FUNCTION_BLOCK Q_Size (* Command change size ( Part 6 - F.18 ) *)
  (* Standard: ISO 11783-6; Description: Copyright (c) 2022 HR Agrartechnik GmbH This program and the accompanying materials are made available under the terms of the Eclipse Public License 2.0 which is available at https://www.eclipse.org/legal/epl-2.0/ SPDX-License-Identifier: EPL-2.0 see Description Tab *)
  (* Version 1.2, 2026-09-05, Franz Höpfinger, HR Agrartechnik GmbH, Implement xScale scaling multiply *)
  (* Version 1.1, 2026-09-05, Franz Höpfinger, HR Agrartechnik GmbH, Add xScale flag *)
  (* Version 1.0, 2022-07-08, Franz Höpfinger, HR Agrartechnik GmbH *)
  PACKAGE isobus::UT::Q;
  IMPORT isobus::UT::Q::const::IDs::ID_NULL;
  (* Documentation:
  Command change size  ( Part 6 - F.18 )
   The Change Size command is used to change the size of an object. A value of 0 for width or height (or both) means that the object size is 0 and the object is not drawn (Annex F.18). The command targets objects that have the sizeable attribute.
   Valid Object IDs
   A sizeable Object ID is valid if it falls within one of the following ISO 11783-6 ID ranges:
    - Container: 3000 – 3999
   - Button: 6000 – 6999
   - InputBooleanField: 7000 – 7999
   - InputStringField: 8000 – 8999
   - InputNumberField: 9000 – 9999
   - InputListField: 10000 – 10999
   - OutputStringField: 11000 – 11999
   - OutputNumberField: 12000 – 12999
   - TypLine: 13000 – 13999
   - TypRectangle: 14000 – 14999
   - TypEllipse: 15000 – 15999
   - TypPolygon: 16000 – 16999
   - Meter: 17000 – 17999
   - LinearBarGraph: 18000 – 18999
   - ArchedBarGraph: 19000 – 19999
   - OutputListObject: 37000 – 37999
   - AnimationObject: 44000 – 44999
    ID_NULL (65535) is not a command target but can be used in INIT to deactivate the FB. Any ID outside these ranges is invalid for commanding.
   Activate / Deactivate
   The FB is deactivated by default. It becomes active when INIT provides a valid sizeable Object ID. Sending INIT with ID_NULL (65535) deactivates the FB again. This toggle can be repeated arbitrarily.
    - INIT + ID_NULL (65535): FB deactivated, STATUS="DEACTIVATED", s16result=VT_E_DEACTIVATED (-40)
   - INIT + valid sizeable ID: FB activated, STATUS="initialized", s16result=VT_E_NO_ERR (0). If a REQ was buffered before, it is executed immediately.
   - INIT + invalid ID: STATUS="ERROR: Invalid Object ID (not a sizeable object)", s16result=VT_E_INVALID_OBJECT_ID (-132)
    REQ Handling
    - REQ before any INIT: Buffered, STATUS="Buffered: INIT not yet completed", s16result=VT_E_NOT_READY (-131)
   - REQ while deactivated (INIT came with NULL or invalid ID): STATUS shows the actual deactivation reason, s16result=VT_E_DEACTIVATED (-40) or VT_E_INVALID_OBJECT_ID (-132)
   - REQ while active: Command sent to VT, result reflected in CNF
    param[in] {objectID, uint16_t}
   Object ID. Use ID_NULL (65535) to deactivate the FB. Use a valid sizeable object ID to activate.
   param[in] {newWidth, uint16_t}
   New width
   param[in] {newHeight, uint16_t}
   New height
   Return Values (s16result):
   int16_t
    - VT_E_NO_ERR (0) - OK
   - VT_E_DEACTIVATED (-40) - FB deactivated (INIT received with ID_NULL)
   - VT_E_INVALID_OBJECT_ID (-132) - Object ID is invalid (not a sizeable object)
   - VT_E_NOT_READY (-131) - Buffered: INIT not yet completed
   - VT_E_OVERFLOW (-6) - buffer overflow
   - VT_E_NOACT (-8) - Command not possible in current state
   - VT_E_NO_INSTANCE (-21) - No VT client available
   - VT_E_ISO_INSTANCE_INVALID (-129) - Identifier for instance (connection) invalid
   - VT_E_NOT_ALIVE (-130) - Identifier for instance valid, but VT Dead.
    Instanz-Eindeutigkeit (Instance Uniqueness)
   Dieser Baustein erfordert Instanz-Eindeutigkeit bezüglich u16ObjId. Es darf im gesamten Programm nur eine Instanz von Q_Size für dieselbe Ziel-Objekt-ID existieren. Eine zweite Instanz auf dieselbe Objekt-ID wird bei INIT deaktiviert (STATUS = "This objID is already in use").
  *)
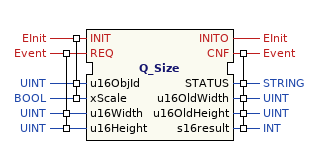
  EVENT_INPUT
    INIT : EInit WITH u16ObjId, xScale; (* Service Initialization *)
    REQ WITH u16Width, u16Height; (* Service Request *)
  END_EVENT
  EVENT_OUTPUT
    INITO : EInit; (* Initialization Confirm *)
    CNF WITH STATUS, s16result, u16OldWidth, u16OldHeight; (* Confirmation of Requested Service *)
  END_EVENT
  VAR_INPUT
    u16ObjId : UINT := ID_NULL; (* Object ID *)
    xScale : BOOL := FALSE; (* FALSE (default) = bypass, send u16Width/u16Height through unchanged. TRUE = scale them by the DM/SKM factor for u16ObjId. *)
    u16Width : UINT; (* New width *)
    u16Height : UINT; (* New height *)
  END_VAR
  VAR_OUTPUT
    STATUS : STRING; (* Service Status *)
    u16OldWidth : UINT; (* Old width *)
    u16OldHeight : UINT; (* Old height *)
    s16result : INT; (* retval see description *)
  END_VAR
END_FUNCTION_BLOCK
